{attribute addProperty BoxType "EK1122-0000-0018"}
{attribute addProperty Id "Beckhoff_EM7xxxsub_EK1100EK1100_179A0949162"}
{attribute addProperty CRC "2132371793"}
{attribute addProperty SizeInBites "16"}
{attribute addProperty SizeInBytes "2"}
TYPE Beckhoff_EM7xxxEK1122_7F196951 EXTENDS EK1122_179A0949 :
STRUCT
	{attribute addProperty Name "Beckhoff_EM7xxxsub_EK1100"}
	Beckhoff_EM7xxxsub_EK1100 : EK1100_179A0949;
END_STRUCT
END_TYPE

(* stored: Version 1.2.0.0, ProductVersion 3.1.4024.9
   DUT Beckhoff_EM7xxxEK1122_7F196951: Id {9751fab9-2b74-4dd6-b010-07f90215d8a9} *)
